// TIA Portal V16 export
// export: Created 2021-11-12T13:31:57.9165134Z, ExportSetting WithDefaults, DisplayName Totally Integrated Automation Portal, DisplayVersion V16 Update 3, DisplayName TIA Portal Version Control Interface, DisplayVersion V16 Update 2, DisplayName TIA Portal Openness, DisplayVersion V16 Update 3, DisplayName SINAMICS Startdrive Advanced, DisplayVersion V16 Update 5, DisplayName SINAMICS Startdrive G130, G150, S120, S150, SINAMICS MV, S210, DisplayVersion V16 Update 5, DisplayName SINAMICS Startdrive G110M, G120, G120C, G120D, G120P, G115D, DisplayVersion V16 Update 5, DisplayName STEP 7 Professional, DisplayVersion V16 Update 3, DisplayName STEP 7 Safety, DisplayVersion V16, DisplayName WinCC UA Professional, DisplayVersion V16 Update 3
DATA_BLOCK "HMI_PARAM_Zone000"   // DB175
{ S7_Optimized_Access := 'TRUE'; DB_Accessible_From_OPC_UA := 'FALSE' }
VERSION : 0.1
// stored: AutoNumber true, DBAccessibleFromOPCUA false, IsOnlyStoredInLoadMemory false, IsRetainMemResEnabled false, IsWriteProtectedInAS false, MemoryReserve 100
   VAR
      Zone000_Mode : "UDT_Zone_Parameter";   // Parameters of zone 000
      StationMEM1_Mode : "UDT_Station_Parameter";   // Parameters of station MEM1
      xxxxx___BinarySensors___xxxxx_1 : Byte;
      "EQ01-BL01" : "UDT_CH_DI_Parameter";   // Hladinový snímač Min LSL 1513 Čerpací jímka 2 (15m3) Hladina OK
      "EQ01-BL02" : "UDT_CH_DI_Parameter";   // Hladinový snímač Max LSL 1514 Čerpací jímka 2 (15m3) Hladina OK
      "EQ01-BL03" : "UDT_CH_DI_Parameter";   // Hladinový snímač Min LSL 1515 Čerpací jímka 2 (5m3) Hladina OK
      "EQ01-BL04" : "UDT_CH_DI_Parameter";   // Hladinový snímač Max LSL 1516 Čerpací jímka 2 (5m3) Hladina OK
      xxxxx___Drives___xxxxx_1 : Byte;
   END_VAR
   VAR RETAIN
      "EQ01-MA01" : "UDT_Drive1_Parameter";   // Pump (P51) / Čerpadlo cirkulace (P31)
      "EQ01-MA02" : "UDT_Drive1_Parameter";   // Pump (P52) / Valve with servomotor (A1417) - draining
      "EQ02-MA01" : "UDT_Drive1_Parameter";   // Pump (P61) / Valve with servomotor (A1417) - draining
      "UC11-TA01" : "UDT_SINAMICS_G120_Parameter";   // Frequence inverter for P51 / Frekvenční měnič ( pro P33)
      "UC11-TA02" : "UDT_SINAMICS_G120_Parameter";   // Frequence inverter for P52 / Frekvenční měnič
      "UC11-TA03" : "UDT_SINAMICS_G120_Parameter";   // Frequence inverter for P61 / Frekvenční měnič
   END_VAR
   VAR
      xxxxx__Alarms__xxxxx { S7_SetPoint := 'True'} : Byte;
      ArchivePeriodicallyBufferWarning : "UDT_DI_Mon_Parameter";
      ArchivePeriodicallyBufferAlarm : "UDT_DI_Mon_Parameter";
      ArchiveItemBufferWarning : "UDT_DI_Mon_Parameter";
      ArchiveItemBufferAlarm : "UDT_DI_Mon_Parameter";
   END_VAR
BEGIN
   "UC11-TA01".RefSpdP2000 := 3000.0;
   "UC11-TA01".RefCurrP2002 := 17.4;
   "UC11-TA01".RefTrqP2003 := 46.91;
   "UC11-TA02".RefSpdP2000 := 3000.0;
   "UC11-TA02".RefCurrP2002 := 17.4;
   "UC11-TA02".RefTrqP2003 := 46.91;
   "UC11-TA03".RefSpdP2000 := 3000.0;
   "UC11-TA03".RefCurrP2002 := 17.4;
   "UC11-TA03".RefTrqP2003 := 46.91;
END_DATA_BLOCK
